FUNCTION_BLOCK ButtonTimerLogic (* Basic Function Block Type *)
  (* Standard: 61499-2 *)
  (* Version 0.0, 5/18/2015, trauscher, nxtControl GmbH, Template *)
  PACKAGE Loytec.Automation;
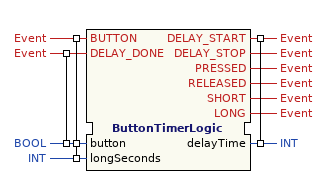
  EVENT_INPUT
    BUTTON WITH button, longSeconds; (* Button event *)
    DELAY_DONE WITH button; (* External delay event *)
  END_EVENT
  EVENT_OUTPUT
    DELAY_START WITH delayTime; (* Start external delay *)
    DELAY_STOP; (* Stop external delay *)
    PRESSED; (* Event when button is pressed *)
    RELEASED; (* Event when button is released *)
    SHORT; (* Event when short press is detected *)
    LONG; (* Event when long press is detected *)
  END_EVENT
  VAR_INPUT
    button : BOOL; (* Button input *)
    longSeconds : INT; (* Time for long press *)
  END_VAR
  VAR_OUTPUT
    delayTime : INT; (* Time for external delay *)
  END_VAR
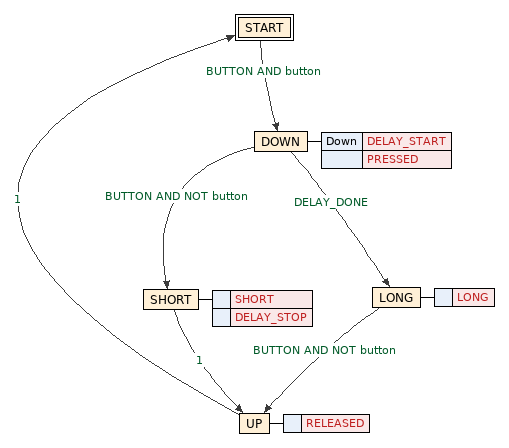
  EC_STATES
    START; (* Initial State *)
    DOWN : Down -> DELAY_START, -> PRESSED;
    UP : -> RELEASED;
    SHORT : -> SHORT, -> DELAY_STOP;
    LONG : -> LONG;
  END_STATES
  EC_TRANSITIONS
    START TO DOWN := BUTTON AND button;
    DOWN TO SHORT := BUTTON AND NOT button;
    UP TO START := 1;
    DOWN TO LONG := DELAY_DONE;
    LONG TO UP := BUTTON AND NOT button;
    SHORT TO UP := 1;
  END_TRANSITIONS
  ALGORITHM Down IN ST:
delayTime := REAL_TO_TIME(longSeconds * 1000.0);
  END_ALGORITHM
END_FUNCTION_BLOCK
